INTERFACE I_MyComponent

PROPERTY SystemErrorPresent : BOOL
GET
END_GET
SET
END_SET
END_PROPERTY

PROPERTY SystemState : E_PMLState
GET
END_GET
SET
END_SET
END_PROPERTY

END_INTERFACE

(* stored: Version 1.1.0.1
   Itf I_MyComponent: Id {8709784e-273d-4e4c-a900-804277c14a47}
   Property SystemErrorPresent: Id {c471a517-367e-4ab9-8a08-8f60e77893a1}
   Get Get: Id {89301abe-b181-4636-a617-ecacc7940fad}
   Set Set: Id {335d9f79-a4eb-4923-a20d-f88d00670403}
   Property SystemState: Id {d609d1e5-e4e2-4903-aef2-7abc0b67e10c}
   Get Get: Id {4647b906-14d7-420e-b551-083ae4c646dc}
   Set Set: Id {c3bd3efd-bb1f-4304-83db-910fdcb6f49f} *)
